INTERFACE I_USINT EXTENDS I_Datatype

PROPERTY PUBLIC Value : REFERENCE TO USINT
GET
END_GET
END_PROPERTY

END_INTERFACE

(* stored: Version 1.1.0.1, ProductVersion 3.1.4024.15
   Itf I_USINT: Id {dcf6164e-b5ba-0e05-0029-3834e64e173f}
   Property Value: Id {c2c0c38e-1a9d-0a84-3b70-9a83e1d81e8f}
   Get Get: Id {f19803be-ca81-050d-3f18-acbd21735195} *)
